TYPE S_PosXY :
STRUCT
	X : LREAL;
	Y : LREAL;
END_STRUCT
END_TYPE

(* stored: Version 1.1.0.1
   DUT S_PosXY: Id {368bd509-1be1-4c78-9720-8535110c0c1a} *)
